// TIA Portal V17 export
// export: Created 2025-01-08T13:55:37.7588729Z, ExportSetting WithDefaults, DisplayName Totally Integrated Automation Portal, DisplayVersion V17, DisplayName TIA Portal Openness, DisplayVersion V17, DisplayName TIA Portal Version Control Interface, DisplayVersion V17, DisplayName SINAMICS Startdrive Advanced, DisplayVersion V17 Update2, DisplayName SINAMICS Startdrive G130, G150, S120, S150, SINAMICS MV, S210, DisplayVersion V17 Update2, DisplayName SINAMICS Startdrive G110M, G120, G120C, G120D, G120P, G115D, DisplayVersion V17 Update2, DisplayName STEP 7 Professional, DisplayVersion V17, DisplayName STEP 7 Safety, DisplayVersion V17, DisplayName WinCC Advanced, DisplayVersion V17
TYPE "HSMMachineParaMask5"
// stored: IsFailsafeCompliant false
   STRUCT
      iRewinderDiameterFull : Bool;
      iMotorLoadLimit : Bool;
      iContourRamp : Bool;
      iEncoderOutPulsPermm : Bool;
      iPLCRackAndSlot : Bool;
      iSliceDistance : Bool;
      iSpliceSpeedReduction : Bool;
      iDownstream : Bool;
      iSpeedFactor : Bool;
      iAcceleration : Bool;
      iSpeedOffset : Bool;
      iMaterialTransportErrorMode : Bool;
      iEncoderFactor : Bool;
      MPARA_I_Reserve_7 : Bool;
      MPARA_I_Reserve_8 : Bool;
      MPARA_I_Reserve_9 : Bool;
   END_STRUCT;
END_TYPE
